TYPE "Sunny_inverter"
VERSION : 0.1
   STRUCT
      InvOpMod : DInt;   // Operating state of the inverter, setpoint
      RemRdy : DInt;   // Put inverter into operation or standby
      "GriMng.VArMod" : DInt;   // Utility grid system services: Selection of procedure for setpoint for reactive power
      "GriMng.WMod" : DInt;   // Utility grid system services: Selection of procedure for setpoint for active power
      ErrClr : DInt;   // Acknowledgment of the present error
      "ErrClr.ProErr" : DInt;   // Acknowledging of safety- relevant errors
      "InvMs.TotVA" : DInt;   // Apparent power, total
      "InvMs.TotW" : DInt;   // Active power, total
      InstFunc : DInt;   // Activation of installation functions
      "InvMs.TotVAr" : DInt;   // Reactive power, total
      "GriMs.Hz" : Real;   // Grid frequency
      ErrLcn : DInt;   // Error location of the present error
      ErrStt : DInt;   // Error status of the inverter
      ErrNo : DInt;   // Error number of the present error
      OpStt : DInt;   // Operating state of the inverter
      WSpt : DInt;   // Active power, setpoint
      VArSpt : DInt;   // Reactive power, setpoint
      PFSpt : Real;   // Power factor cos (phi), setpoint
      WAval : Real;   // Currently available active power
      VArAval : Real;   // Currently available reactive power
      PwrOffReas : DInt;   // Current cause of inverter disconnection
      DrtStt : DInt;   // Derating status
      WSpt_pct : Int;   // UID2 addr 23 - WSpt % FIX2 raw (100% = 10000)
      VArSpt_pct : Int;   // UID2 addr 22 - VArSpt % FIX2 raw (100% = 10000)
      PF_cos : Word;   // UID2 addr 24 - PF magnitude U16 FIX4 (cos_phi x 10000)
      PF_excitation : DWord;   // UID2 addr 25 - PF direction ENUM (1041=OE, 1042=UE)
   END_STRUCT;

END_TYPE

